Universal Robots PolyScope program: step4d_circle_detsearch_attitude_v1.urp

Program step4d_circle_detsearch_attitude_v1 (installation=default directory=/programs/andyl/kunwei/step4/step4abcd createdIn=5.11.9.1010452 lastSavedIn=5.11.9.1010452 robotSerialNumber=20225200364)
Calibrated DH parameters: a=[0.00002, -0.569483, -0.54992, -0.00001, -0.000036, 0]; d=[0.180894, -146.691669, 192.918669, -46.053088, 0.119778, 0.115602]; alpha=[1.571425, -0.001534, 0.003359, 1.568739, -1.571477, 0]; deltaTheta=[0, 0.376258, -0.101074, -0.275185, -0.000002, 0]
Robot Program (runOnlyOnce=true)
  Script file /programs/andyl/kunwei/step4/step4abcd/step4d_circle_detsearch_attitude_v1.script
    | # Step4d contact circle v1: deterministic contact search, full-circle Cartesian speedl, Z force admittance, and velocity attitude admittance.
    | # VERSION: 2026-06-08T1650HKT_STEP4D_CIRCLE_DETSEARCH_ATTITUDE_V1
    | # GENERATED_AT_LOCAL: 2026-06-08T16:50:19+0800
    | # BEHAVIOR: wait for Kunwei bridge; align to old reference orientation; move to
    | # Step4d circle-start XY derived from the middle half of the old contact path;
    | # do bounded Z prep instead of blindly returning to contact Z + 100 mm. If current Z is already 30-100 mm above known contact,
    | # keep it. Then search downward at 15 mm/s until 10 mm above known contact,
    | # 3 mm/s near the surface, using 2 ms speedl holds and no force-admittance
    | # downward command before confirmed contact. Small-force contact is accepted
    | # only in the near zone; far-zone unexpected contact stops and auto-homes. The
    | # first 0.10 s of circle control uses 10 ms speedl holds, then circle control
    | # switches to 1 ms holds. The circle stage commands Cartesian twist, so UR still owns IK.
    | # Circle-stage normal Z correction targets signed Fz ~= -target_force_abs, where the bridge
    | # normally writes target_force_abs=5 N into input register 29. Attitude admittance
    | # uses lateral force and Mx/My as a bounded wx/wy velocity correction.
    | # Raw contact triggers and safety guards remain unfiltered; only controller
    | # normal-velocity input uses a light force filter. No UR zero_ftsensor, no
    | # Kunwei tare/config write, no TCP/payload write, and no output register 34.
    | # Frequency contract: Kunwei raw may be about 1 kHz; RTDE handoff is requested
    | # at 500 Hz; deterministic search uses 2 ms speedl holds; line control
    | # switches to 1 ms holds after 0.10 s, but both phases must be measured before
    | # calling them 500 Hz authority. On recoverable stops, retract 10 mm upward
    | # and then return to the TP-start home pose while preserving the true stop reason.
    | 
    | def codex_abs(x):
    |   if x < 0.0:
    |     return -x
    |   end
    |   return x
    | end
    | 
    | def codex_clamp(x, lo, hi):
    |   if x < lo:
    |     return lo
    |   elif x > hi:
    |     return hi
    |   end
    |   return x
    | end
    | 
    | def codex_wait_for_sensor_ok(timeout_s):
    |   local dt = 0.002
    |   local t = 0.0
    |   while t < timeout_s:
    |     if read_input_float_register(27) > 0.5:
    |       return True
    |     end
    |     sync()
    |     t = t + dt
    |   end
    |   return False
    | end
    | 
    | def codex_wait_for_fresh_heartbeat(timeout_s):
    |   local dt = 0.002
    |   local t = 0.0
    |   local initial_heartbeat = read_input_float_register(26)
    |   local current_heartbeat = initial_heartbeat
    |   while t < timeout_s:
    |     current_heartbeat = read_input_float_register(26)
    |     write_output_float_register(26, current_heartbeat)
    |     write_output_float_register(35, 20.5)
    |     if read_input_float_register(27) > 0.5 and current_heartbeat != initial_heartbeat:
    |       return True
    |     end
    |     sync()
    |     t = t + dt
    |   end
    |   return False
    | end
    | 
    | def codex_step2_guard_stop_reason():
    |   local normal_force = read_input_float_register(24)
    |   local force_norm = read_input_float_register(25)
    |   local sensor_ok = read_input_float_register(27)
    |   local stop_request = read_input_float_register(28)
    |   local torque_norm = read_input_float_register(30)
    |   if sensor_ok < 0.5:
    |     return 3.0
    |   elif stop_request > 0.5:
    |     return 4.0
    |   elif codex_abs(normal_force) > 20.0:
    |     return 5.0
    |   elif force_norm > 50.0:
    |     return 6.0
    |   elif torque_norm > 0.6:
    |     return 7.0
    |   end
    |   return 0.0
    | end
    | 
    | def codex_should_auto_home(stop_reason):
    |   if stop_reason == 1.0:
    |     return True
    |   elif stop_reason == 2.0:
    |     return True
    |   elif stop_reason == 4.0:
    |     return True
    |   elif stop_reason == 8.0:
    |     return True
    |   elif stop_reason == 9.0:
    |     return True
    |   elif stop_reason == 10.0:
    |     return True
    |   elif stop_reason == 12.0:
    |     return True
    |   elif stop_reason == 13.0:
    |     return True
    |   end
    |   return False
    | end
    | 
    | def codex_write_echo(stop_reason, progress_m, correction_m, commanded_z_m_s):
    |   write_output_float_register(24, read_input_float_register(24))
    |   write_output_float_register(25, read_input_float_register(25))
    |   write_output_float_register(26, read_input_float_register(26))
    |   write_output_float_register(27, read_input_float_register(27))
    |   write_output_float_register(28, read_input_float_register(28))
    |   write_output_float_register(29, read_input_float_register(29))
    |   write_output_float_register(30, stop_reason)
    |   write_output_float_register(31, progress_m)
    |   write_output_float_register(32, correction_m)
    |   write_output_float_register(33, commanded_z_m_s)
    | end
    | 
    | def codex_step4d_circle_detsearch_attitude():
    |   local ux = 0.679764156
    |   local uy = -0.733430768
    |   local entry_x = 0.457390615
    |   local entry_y = 0.215059119
    |   local old_contact_z = 0.020279919
    |   local entry_z = old_contact_z + 0.100
    |   local ref_rx = 3.141572714
    |   local ref_ry = -0.000026465
    |   local ref_rz = -0.000024158
    |   local approach_speed_m_s = 0.080
    |   local approach_z_speed_m_s = 0.080
    |   local search_accel_m_s2 = 0.300
    |   local search_hold_s = 0.002
    |   local max_search_down_m = 0.110
    |   local stale_limit_s = 0.100
    |   local search_runtime_limit_s = 65.0
    |   local tangent_speed_m_s = 0.005
    |   local path_length_m = 0.09987123
    |   local line_accel_m_s2 = 0.300
    |   local circle_radius_m = 0.015895
    |   local two_pi = 6.283185307
    |   local circle_direction = 1
    |   local circle_perp_x = 0.733430768
    |   local circle_perp_y = 0.679764156
    |   local circle_xy_p_gain_m_s_per_m = 3.0
    |   local circle_xy_velocity_limit_m_s = 0.003
    |   local angular_velocity_limit_rad_s = 0.030
    |   local attitude_force_gain_rad_s = 0.040
    |   local attitude_torque_gain_rad_s_per_nm = 0.050
    |   local attitude_filter_alpha = 0.20
    |   local max_attitude_error_proxy_rad = 0.35
    |   local line_hold_s = 0.010
    |   local line_hold_fast_s = 0.001
    |   local line_fast_after_s = 0.100
    |   local line_runtime_limit_s = 30.0
    |   local target_force_abs_default_n = 5.0
    |   local target_force_ramp_start_n = 1.0
    |   local target_force_ramp_s = 2.0
    |   local normal_velocity_p_gain = 0.0006
    |   local normal_velocity_i_gain = 0.00008
    |   local normal_velocity_limit_m_s = 0.005
    |   local normal_filter_alpha = 0.70
    |   local integral_error_limit_n_s = 10.0
    |   local short_retract_z_m = 0.010
    |   local short_retract_speed_m_s = 0.020
    |   local home_return_speed_m_s = 0.080
    |   local stop_reason = 0.0
    |   local contact_triggered = 0
    |   local max_observed_stale_s = 0.0
    |   local final_progress_m = 0.0
    | 
    |   local home_pose = get_actual_tcp_pose()
    | 
    |   textmsg("codex step4d version 2026-06-08T1650HKT_STEP4D_CIRCLE_DETSEARCH_ATTITUDE_V1 start circle_detsearch_attitude_v1")
    |   write_output_float_register(35, 20.0)
    |   codex_write_echo(0.0, 0.0, 0.0, 0.0)
    | 
    |   if not codex_wait_for_fresh_heartbeat(30.0):
    |     stop_reason = 3.0
    |   end
    | 
    |   if stop_reason == 0.0:
    |     write_output_float_register(35, 21.0)
    |     local p0 = get_actual_tcp_pose()
    |     local reference_orientation_pose = p[p0[0], p0[1], p0[2], ref_rx, ref_ry, ref_rz]
    |     movel(reference_orientation_pose, a=0.030, v=approach_speed_m_s, r=0.0)
    |     stopl(0.5)
    |     write_output_float_register(35, 22.0)
    |     local p1 = get_actual_tcp_pose()
    |     local entry_xy_pose = p[entry_x, entry_y, p1[2], ref_rx, ref_ry, ref_rz]
    |     movel(entry_xy_pose, a=0.030, v=approach_speed_m_s, r=0.0)
    |     stopl(0.5)
    |     write_output_float_register(35, 23.0)
    |     local p2 = get_actual_tcp_pose()
    |     local max_entry_z = old_contact_z + 0.100
    |     local min_entry_z = old_contact_z + 0.030
    |     local bounded_entry_z = p2[2]
    |     if bounded_entry_z > max_entry_z:
    |       bounded_entry_z = max_entry_z
    |     elif bounded_entry_z < min_entry_z:
    |       bounded_entry_z = min_entry_z
    |     end
    |     if codex_abs(bounded_entry_z - p2[2]) > 0.002:
    |       local entry_pose = p[entry_x, entry_y, bounded_entry_z, ref_rx, ref_ry, ref_rz]
    |       movel(entry_pose, a=0.030, v=approach_z_speed_m_s, r=0.0)
    |       stopl(0.5)
    |     end
    |     sleep(0.20)
    |     stop_reason = codex_step2_guard_stop_reason()
    |   end
    | 
    |   if stop_reason == 0.0:
    |     write_output_float_register(35, 24.0)
    |     local search_start = get_actual_tcp_pose()
    |     local last_heartbeat = read_input_float_register(26)
    |     local stale_s = 0.0
    |     local t = 0.0
    |     local search_far_speed_m_s = -0.015
    |     local search_near_speed_m_s = -0.003
    |     local search_near_zone_m = 0.010
    |     local contact_normal_force_n = -1.0
    |     local contact_force_norm_n = 1.5
    |     local far_unexpected_normal_force_n = -5.0
    |     local far_unexpected_force_norm_n = 5.0
    |     local near_contact = 0
    |     local commanded_search_z = search_far_speed_m_s
    |     while stop_reason == 0.0:
    |       local heartbeat = read_input_float_register(26)
    |       local normal_force = read_input_float_register(24)
    |       local force_norm = read_input_float_register(25)
    |       local pose_now = get_actual_tcp_pose()
    |       local search_depth_m = search_start[2] - pose_now[2]
    |       local height_above_known_contact_m = pose_now[2] - old_contact_z
    | 
    |       if heartbeat == last_heartbeat:
    |         stale_s = stale_s + search_hold_s
    |         if stale_s > max_observed_stale_s:
    |           max_observed_stale_s = stale_s
    |         end
    |       else:
    |         stale_s = 0.0
    |         last_heartbeat = heartbeat
    |       end
    | 
    |       write_output_float_register(35, 24.0)
    |       if height_above_known_contact_m <= search_near_zone_m:
    |         if normal_force <= contact_normal_force_n or force_norm > contact_force_norm_n:
    |           near_contact = 1
    |           write_output_float_register(35, 24.8)
    |         end
    |       elif normal_force <= far_unexpected_normal_force_n or force_norm > far_unexpected_force_norm_n:
    |         stop_reason = 13.0
    |       end
    | 
    |       if stop_reason == 0.0 and stale_s > stale_limit_s:
    |         stop_reason = 2.0
    |       elif stop_reason == 0.0:
    |         stop_reason = codex_step2_guard_stop_reason()
    |       end
    | 
    |       if stop_reason == 0.0:
    |         if near_contact == 1:
    |           contact_triggered = 1
    |           stop_reason = 11.0
    |           codex_write_echo(stop_reason, max_observed_stale_s, search_depth_m, 0.0)
    |         elif search_depth_m >= max_search_down_m:
    |           stop_reason = 8.0
    |         elif t >= search_runtime_limit_s:
    |           stop_reason = 10.0
    |         else:
    |           if height_above_known_contact_m > search_near_zone_m:
    |             commanded_search_z = search_far_speed_m_s
    |           else:
    |             commanded_search_z = search_near_speed_m_s
    |           end
    |           codex_write_echo(stop_reason, max_observed_stale_s, search_depth_m, commanded_search_z)
    |           speedl([0.0, 0.0, commanded_search_z, 0.0, 0.0, 0.0], search_accel_m_s2, search_hold_s)
    |           t = t + search_hold_s
    |         end
    |       end
    |     end
    |     stopl(0.5)
    | 
    |     if stop_reason == 8.0:
    |       write_output_float_register(35, 28.0)
    |       local p_end = get_actual_tcp_pose()
    |       local retract_pose = p[p_end[0], p_end[1], entry_z, p_end[3], p_end[4], p_end[5]]
    |       movel(retract_pose, a=0.030, v=0.005, r=0.0)
    |       stopl(0.5)
    |     end
    |   end
    | 
    |   if contact_triggered == 1:
    |     stop_reason = 0.0
    |   end
    | 
    |   if stop_reason == 0.0:
    |     write_output_float_register(35, 25.0)
    |     local circle_start_pose = get_actual_tcp_pose()
    |     local last_heartbeat2 = read_input_float_register(26)
    |     local stale_s2 = 0.0
    |     local t2 = 0.0
    |     local theta = 0.0
    |     local filtered_normal_force = read_input_float_register(24)
    |     local filtered_fx = read_input_float_register(31)
    |     local filtered_fy = read_input_float_register(32)
    |     local filtered_mx = read_input_float_register(34)
    |     local filtered_my = read_input_float_register(35)
    |     local integral_error = 0.0
    |     while stop_reason == 0.0:
    |       if t2 >= line_fast_after_s:
    |         line_hold_s = line_hold_fast_s
    |       end
    |       local raw_normal_force = read_input_float_register(24)
    |       local heartbeat2 = read_input_float_register(26)
    |       local requested_target_force_abs = read_input_float_register(29)
    |       local pose_line = get_actual_tcp_pose()
    |       local progress_m = theta * circle_radius_m
    |       local correction_m = pose_line[2] - circle_start_pose[2]
    |       final_progress_m = progress_m
    | 
    |       if requested_target_force_abs < 0.1:
    |         requested_target_force_abs = target_force_abs_default_n
    |       end
    |       local target_force_ramp_alpha = codex_clamp(t2 / target_force_ramp_s, 0.0, 1.0)
    |       local target_force_abs = target_force_ramp_start_n + (requested_target_force_abs - target_force_ramp_start_n) * target_force_ramp_alpha
    |       if requested_target_force_abs < target_force_ramp_start_n:
    |         target_force_abs = requested_target_force_abs
    |       end
    | 
    |       filtered_normal_force = normal_filter_alpha * raw_normal_force + (1.0 - normal_filter_alpha) * filtered_normal_force
    |       local force_error = target_force_abs + filtered_normal_force
    |       integral_error = codex_clamp(integral_error + force_error * line_hold_s, -integral_error_limit_n_s, integral_error_limit_n_s)
    |       local normal_velocity = 0.0 - codex_clamp(normal_velocity_p_gain * force_error + normal_velocity_i_gain * integral_error, -normal_velocity_limit_m_s, normal_velocity_limit_m_s)
    | 
    |       local fx_n = read_input_float_register(31)
    |       local fy_n = read_input_float_register(32)
    |       local mx_nm = read_input_float_register(34)
    |       local my_nm = read_input_float_register(35)
    |       filtered_fx = attitude_filter_alpha * fx_n + (1.0 - attitude_filter_alpha) * filtered_fx
    |       filtered_fy = attitude_filter_alpha * fy_n + (1.0 - attitude_filter_alpha) * filtered_fy
    |       filtered_mx = attitude_filter_alpha * mx_nm + (1.0 - attitude_filter_alpha) * filtered_mx
    |       filtered_my = attitude_filter_alpha * my_nm + (1.0 - attitude_filter_alpha) * filtered_my
    |       local force_tilt_x = codex_clamp(filtered_fy / target_force_abs, -max_attitude_error_proxy_rad, max_attitude_error_proxy_rad)
    |       local force_tilt_y = codex_clamp(0.0 - filtered_fx / target_force_abs, -max_attitude_error_proxy_rad, max_attitude_error_proxy_rad)
    |       local angular_x = codex_clamp(attitude_force_gain_rad_s * force_tilt_x + attitude_torque_gain_rad_s_per_nm * filtered_mx, -angular_velocity_limit_rad_s, angular_velocity_limit_rad_s)
    |       local angular_y = codex_clamp(attitude_force_gain_rad_s * force_tilt_y + attitude_torque_gain_rad_s_per_nm * filtered_my, -angular_velocity_limit_rad_s, angular_velocity_limit_rad_s)
    | 
    |       local sin_theta = sin(theta)
    |       local cos_theta = cos(theta)
    |       local e1x = circle_direction * circle_perp_x
    |       local e1y = circle_direction * circle_perp_y
    |       local desired_x = circle_start_pose[0] + circle_radius_m * (1.0 - cos_theta) * ux + circle_radius_m * sin_theta * e1x
    |       local desired_y = circle_start_pose[1] + circle_radius_m * (1.0 - cos_theta) * uy + circle_radius_m * sin_theta * e1y
    |       local tangent_vx = tangent_speed_m_s * (sin_theta * ux + cos_theta * e1x)
    |       local tangent_vy = tangent_speed_m_s * (sin_theta * uy + cos_theta * e1y)
    |       local correction_vx = codex_clamp(circle_xy_p_gain_m_s_per_m * (desired_x - pose_line[0]), -circle_xy_velocity_limit_m_s, circle_xy_velocity_limit_m_s)
    |       local correction_vy = codex_clamp(circle_xy_p_gain_m_s_per_m * (desired_y - pose_line[1]), -circle_xy_velocity_limit_m_s, circle_xy_velocity_limit_m_s)
    |       local command_vx = tangent_vx + correction_vx
    |       local command_vy = tangent_vy + correction_vy
    | 
    |       if heartbeat2 == last_heartbeat2:
    |         stale_s2 = stale_s2 + line_hold_s
    |       else:
    |         stale_s2 = 0.0
    |         last_heartbeat2 = heartbeat2
    |       end
    | 
    |       codex_write_echo(stop_reason, progress_m, correction_m, normal_velocity)
    | 
    |       if stale_s2 > stale_limit_s:
    |         stop_reason = 2.0
    |       else:
    |         stop_reason = codex_step2_guard_stop_reason()
    |       end
    | 
    |       if stop_reason == 0.0:
    |         if codex_abs(correction_m) > 0.008:
    |           stop_reason = 8.0
    |         elif progress_m < -0.003 or progress_m > path_length_m + 0.003:
    |           stop_reason = 9.0
    |         elif t2 >= line_runtime_limit_s:
    |           stop_reason = 10.0
    |         elif theta >= two_pi:
    |           stop_reason = 1.0
    |         else:
    |           speedl([command_vx, command_vy, normal_velocity, angular_x, angular_y, 0.0], line_accel_m_s2, line_hold_s)
    |           t2 = t2 + line_hold_s
    |           theta = theta + tangent_speed_m_s * line_hold_s / circle_radius_m
    |         end
    |       end
    |     end
    |     stopl(0.5)
    |   end
    |   if codex_should_auto_home(stop_reason):
    |     write_output_float_register(35, 26.0)
    |     local short_retract_start = get_actual_tcp_pose()
    |     local short_retract_pose = p[short_retract_start[0], short_retract_start[1], short_retract_start[2] + short_retract_z_m, short_retract_start[3], short_retract_start[4], short_retract_start[5]]
    |     codex_write_echo(stop_reason, final_progress_m, short_retract_z_m, 0.0)
    |     movel(short_retract_pose, a=0.030, v=short_retract_speed_m_s, r=0.0)
    |     stopl(0.5)
    |     write_output_float_register(35, 27.0)
    |     codex_write_echo(stop_reason, final_progress_m, short_retract_z_m, 0.0)
    |     movel(home_pose, a=0.030, v=home_return_speed_m_s, r=0.0)
    |     stopl(0.5)
    |   end
    | 
    |   write_output_float_register(30, stop_reason)
    |   write_output_float_register(31, max_observed_stale_s)
    |   write_output_float_register(35, 29.0)
    |   textmsg("codex step4d version 2026-06-08T1650HKT_STEP4D_CIRCLE_DETSEARCH_ATTITUDE_V1 stop reason:", stop_reason)
    | end
    | 
    | codex_step4d_circle_detsearch_attitude()
